// TwinCAT 3 PLC project PLC
// ProgramVersion: 3.1.4024.0
// project tree:
//   / GVL.TcGVL, POU.TcPOU, POU_1.TcPOU
// I/O:
//   DEVICE Device 1 (EtherCAT), AmsNetId 10.10.10.212.2.1

// ---- GVL.TcGVL
{attribute 'qualified_only'}
VAR_GLOBAL
END_VAR

// ---- POU.TcPOU
FUNCTION_BLOCK POU
VAR_INPUT
END_VAR
VAR_OUTPUT
END_VAR
VAR
	a: INT;
	b: INT;
END_VAR

a := a+b;

END_FUNCTION_BLOCK

// ---- POU_1.TcPOU
PROGRAM POU_1
VAR
END_VAR

END_PROGRAM
